PROGRAM Main
VAR
	io_TestSuite : IO_TestSuite;
END_VAR

TcUnit.Run();

END_PROGRAM

(* stored: Version 1.1.0.1, ProductVersion 3.1.4024.12
   POU Main: Id {9fe10dc8-5bf9-09d9-1e39-a2aabc9c3ea3}, SpecialFunc None *)
